TYPE MotorOutputVariables :
STRUCT
	Coil : BOOL;
END_STRUCT
END_TYPE

(* stored: Version 1.1.0.1, ProductVersion 3.1.4024.9
   DUT MotorOutputVariables: Id {fe1dead6-671e-4cd2-ad5c-960ac18d3dd4} *)
